FUNCTION mySign : int
VAR_INPUT
	 a:LREAL;
END_VAR
VAR
END_VAR

 IF (a < 0) THEN mySign:= -1;
    ELSIF (a>0) THEN mySign:= 1;
    ELSE mySign:= 0;
	
	END_IF

END_FUNCTION

(* stored: Version 1.1.0.1, ProductVersion 3.1.4024.12
   POU mySign: Id {7d725517-371b-41c0-ab01-a0e68f62073c}, SpecialFunc None *)
